FUNCTION_BLOCK STARTandSTOP
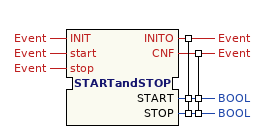
  EVENT_INPUT
    INIT;
    start;
    stop;
  END_EVENT
  EVENT_OUTPUT
    INITO WITH START, STOP;
    CNF WITH START, STOP;
  END_EVENT
  VAR_OUTPUT
    START : BOOL;
    STOP : BOOL;
  END_VAR
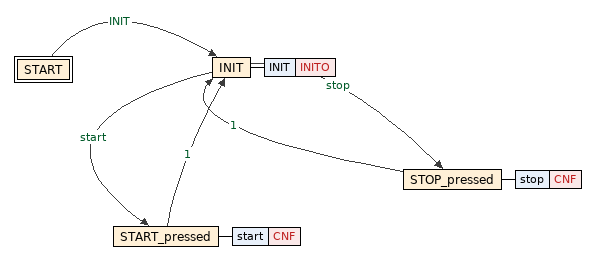
  EC_STATES
    START;
    INIT : INIT -> INITO;
    START_pressed : start -> CNF;
    STOP_pressed : stop -> CNF;
  END_STATES
  EC_TRANSITIONS
    START TO INIT := INIT;
    START_pressed TO INIT := 1;
    STOP_pressed TO INIT := 1;
    INIT TO START_pressed := start;
    INIT TO STOP_pressed := stop;
  END_TRANSITIONS
  ALGORITHM INIT IN ST:
START := FALSE;&#38;#10;STOP := FALSE;&#38;#10;
  END_ALGORITHM
  ALGORITHM start IN ST:
START := TRUE;&#38;#10;
  END_ALGORITHM
  ALGORITHM stop IN ST:
STOP := TRUE;&#38;#10;
  END_ALGORITHM
END_FUNCTION_BLOCK
